(* Logix 5000 project; controller HW3 vendor 1 type 14 code 92 rev 28.11; software revision 28.00 *)

TASK MainTask (continuous, watchdog 500 ms) : MainProgram

MODULES
   Local : vendor 1 type 14 code 92 (ICP 0, rev 28.11)
      Digital_IN : 1756-IB16 (ICP 2, rev 3.1, Input RPI 20 ms)
      Digital_OUT : vendor 1 type 7 code 18 (ICP 4, rev 3.1, Output RPI 20 ms)
      Analog_IN : 1756-IF8 (ICP 6, rev 1.1, Input RPI 100 ms)
END_MODULES

PROGRAM MainProgram   (* main routine MainRoutine *)
VAR
   CT1 : COUNTER; {access Read Only}   // Counter 1
   HV : ALIAS FOR Local:6:I.Ch0Data;   // Height Voltage
   M1 : ALIAS FOR Local:4:O.Data.0;   // Conveyor Motor
   PB1 : ALIAS FOR Local:2:I.Data.0;   // Push Button 1
   PS1 : ALIAS FOR Local:2:I.Data.1;   // Photo Switch 1
   TM1 : TIMER := (PRE := 1);   // Timer 1
   TOG1L : ALIAS FOR Local:2:I.Data.3;   // Toggle Switch 1: Lower Position
   TOG1U : ALIAS FOR Local:2:I.Data.2;   // Toggle Switch 1: Upper Position
   TOG2L : ALIAS FOR Local:2:I.Data.5;   // Toggle Switch 2: Lower Position
   TOG2U : ALIAS FOR Local:2:I.Data.4;   // Toggle Switch 2: Upper Position
   TP : DINT;   // Passage of Time Photo Switch is Activated
   YL : ALIAS FOR Local:4:O.Data.1;   // Yellow Light
END_VAR

ROUTINE MainRoutine   (* ladder *)
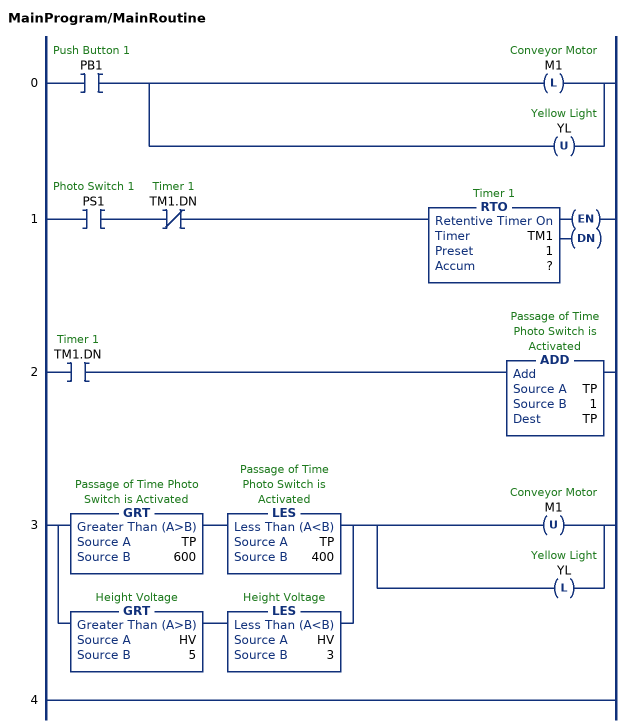
   0: XIC(PB1)[OTL(M1) ,OTU(YL) ];
   1: XIC(PS1)XIO(TM1.DN)RTO(TM1,?,?);
   2: XIC(TM1.DN)ADD(TP,1,TP);
   3: [GRT(TP,600) LES(TP,400) ,GRT(HV,5) LES(HV,3) ][OTU(M1) ,OTL(YL) ];
   4: ;
END_ROUTINE
END_PROGRAM
